PROGRAM MAIN
VAR
    pidSuite : FB_PidTests;
    rbSuite  : FB_RingBufferTests;
    strSuite : FB_StringTests;
END_VAR

TcUnit.RUN_IN_SEQUENCE();

END_PROGRAM

(* stored: Version 1.1.0.1
   POU MAIN: Id {7794d574-dac1-40b7-b376-bf7ff0ac4646}, SpecialFunc None *)
